Staubli VAL3: default.pjx

Parameters version=s8.10.2cs9_BS1991 stackSize=5000 millimeterUnit=true
Program file=start.pgx
Program file=stop.pgx
Data file=default.dtx
